// TIA Portal V16 export
// export: Created 2024-05-16T13:10:21.6108295Z, ExportSetting WithDefaults, DisplayName Totally Integrated Automation Portal, DisplayVersion V16, DisplayName TIA Portal Version Control Interface, DisplayVersion V16, DisplayName TIA Portal Openness, DisplayVersion V16, DisplayName STEP 7 Professional, DisplayVersion V16, DisplayName STEP 7 Safety, DisplayVersion V16, DisplayName WinCC Professional, DisplayVersion V16
DATA_BLOCK "DB22001_Dy_InstAnalogRead"   // DB22001
TITLE = Dynamic DB [INSTRUMENTATION] — Analog Instrument Read, Scale and Monitor
{ S7_Optimized_Access := 'TRUE' }
AUTHOR : M_Gledhill
FAMILY : Instrumentation
NAME : Dy_InstAnalogRead
VERSION : 3.0
// PRACTICAL SERIES AUTOMATION LIBRARY (PAL)   —   COPYRIGHT 2020 – M. GLEDHILL (MIT LICENCE)
//                   ———— ◆ ————
// FULL ONLINE DOCUMENTATION IS AVAILABLE AT: https://practicalseries.com/2001-pal/index.html
// stored: AutoNumber false, DBAccessibleFromOPCUA true, IsOnlyStoredInLoadMemory false, IsRetainMemResEnabled false, IsWriteProtectedInAS false, MemoryReserve 100
   VAR
      _DB_Header { ExternalAccessible := 'False'; ExternalVisible := 'False'; ExternalWritable := 'False'} : Array[0..79] of Bool;   // Dynamic DB [INSTRUMENTATION] — Analog Instrument Read, Scale and Monitor
      __________0000_0 { ExternalAccessible := 'False'; ExternalVisible := 'False'; ExternalWritable := 'False'} : Bool := false;
      __________0000_1 { ExternalAccessible := 'False'; ExternalVisible := 'False'; ExternalWritable := 'False'} : Bool := false;   // ▀▀▀▀ DB CURRENT REVISION
      revInfo { ExternalWritable := 'False'; S7_SetPoint := 'True'} : "UT01000_St_SysRevision";   // Revision information
      __________0010_0 { ExternalAccessible := 'False'; ExternalVisible := 'False'; ExternalWritable := 'False'} : Bool := false;
      __________0010_1 { ExternalAccessible := 'False'; ExternalVisible := 'False'; ExternalWritable := 'False'} : Bool := false;   // ▀▀▀▀ ANALOG INSTRUMENTS
      FIC101 { S7_SetPoint := 'True'} : "UT22001_Dy_InstAnalogRead";   // Filter 1 outlet flow
   END_VAR
BEGIN
   // _DB_Header[0] : ▄▄▄▄▄▄▄▄▄▄▄▄▄▄▄▄▄▄▄▄▄▄▄▄▄▄▄▄▄▄▄▄▄ ＳＴＡＮＤＡＲＤ ▄▄
   // _DB_Header[2] : TITLE: INSTRUMENTATION — ANALOG INSTRUMENT READ, SCALE AND MONITOR
   // _DB_Header[4] : ▀▀▀▀▀▀▀▀▀▀▀▀▀▀▀▀▀▀▀▀▀▀▀▀▀▀▀▀▀▀▀▀▀▀▀▀▀▀▀▀▀▀▀▀
   // _DB_Header[5] : TYPE: DYNAMIC
   // _DB_Header[6] : ▄▄▄▄▄▄▄▄▄▄▄▄▄▄▄▄▄▄▄▄▄▄▄▄▄▄▄▄▄▄▄▄▄▄▄▄▄▄▄▄▄▄▄▄
   // _DB_Header[8] : This is the dynamic data block associated with the standard analog instrument read
   // _DB_Header[9] : block:
   // _DB_Header[10] : FC02001_StdInstAnalog
   // _DB_Header[12] : The dynamic data holds the current scaled value of the instrument, along with
   // _DB_Header[13] : any alarms, warnings or faults.
   // _DB_Header[15] : Each instrument is given the user data type:
   // _DB_Header[16] : UT22001_Dy_InstAnalog
   // _DB_Header[17] : This holds the full set of static configuration data for the instrument.
   // _DB_Header[19] : ━━━ ⬙⬙⬙⬙⬙⬙ ━━━
   // _DB_Header[21] : ▄▄▄▄▄▄▄▄▄▄▄▄▄▄▄▄▄▄▄▄▄▄▄▄▄▄▄▄▄▄▄▄▄▄▄▄▄▄▄▄▄▄▄▄
   // _DB_Header[22] : MODIFICATION HISTORY
   // _DB_Header[24] : This is a summary of the recent software modifications made to this block (most recent at top)
   // _DB_Header[26] : ―――――――――――――――――――――――――――――――――――――――――――
   // _DB_Header[27] : DATE REVISION MASTER BRANCH DEV
   // _DB_Header[28] : (nnn.amm) COMMIT TAG (Base ---> Merge) BRANCH Author
   // _DB_Header[29] : ———————————————————————————————————————————
   // _DB_Header[30] : 2024.05.16 003.000 D0017A-000.105 D0017 D0018 None M. Gledhill
   // _DB_Header[31] : FC02001 — RELEASED FOR USE
   // _DB_Header[32] : Merge back to master branch
   // _DB_Header[34] : 2024.05.11 002.801 D0017A-000.104 D0017 N/A D017A M. Gledhill
   // _DB_Header[35] : RAW_ANALOG changed to AI_RAW_SIGNAL
   // _DB_Header[36] : AI_RAW_DATA and AI_SCALE_DATA added and
   // _DB_Header[37] : copied to DYNAMIC_DATA (see db00801 SMDS)
   // _DB_Header[39] : 2022.04.16 002.000 D0011 D0010 D0011 None M. Gledhill
   // _DB_Header[40] : FC02001 — RELEASED FOR USE
   // _DB_Header[41] : Merge back to master branch
   // _DB_Header[43] : 2022.04.11 001.801 D0010A-000.801 D0010 N/A D010A M. Gledhill
   // _DB_Header[44] : Released for test (SCV)
   // _DB_Header[46] : 2022.04.08 001.102 D0010A-000.104 D0010 N/A D010A M. Gledhill
   // _DB_Header[47] : Comments updated
   // _DB_Header[49] : 2022.04.05 001.101 D0010A-000.103 D0010 N/A D010A M. Gledhill
   // _DB_Header[50] : Over and under range based on scaled signal
   // _DB_Header[51] : INFO_TYPE, cal_OR_Abs and cal_UR_Abs added
   // _DB_Header[52] : Comments updated and standardised
   // _DB_Header[53] : UDT variable names standardised
   // _DB_Header[55] : 2021.05.26 001.000 D0008 D0006 D0008 None M. Gledhill
   // _DB_Header[56] : FC02001 — RELEASED FOR USE
   // _DB_Header[57] : Merge back to master branch
   // _DB_Header[59] : 2021.05.24 000.801 D0006B-000.801 D0006 N/A D0006B M. Gledhill
   // _DB_Header[60] : FC02001 — Released for SMT
   // _DB_Header[62] : 2021.05.18 000.101 D0006B-000.101 D0006 N/A D0006B M. Gledhill
   // _DB_Header[63] : FC02001 Migration to VCS
   // _DB_Header[64] : ———————————————————————————————————————————
   // _DB_Header[65] : Where: nnn = Major revision
   // _DB_Header[66] : a = Type (1-7 Development, 8 Proving, 9 Qualification, 0 Release)
   // _DB_Header[67] : mm = Minor revision (must be 00 if a = 0)
   // _DB_Header[68] : Block properties version number should be set to nn.a (only one decimal place)
   // _DB_Header[70] : ██████████████ █ █ █ █ END █ █ █ █ ██████████████
   revInfo.REV_BLOCK := 'DB22001';
   revInfo.REV_NUMBER := '003.000';
   revInfo.REV_DATE := '2024-05-16';
   revInfo.REV_AUTHOR := 'M. Gledhill';
   FIC101.revInfo.REV_BLOCK := 'DB22001';
   FIC101.revInfo.REV_NUMBER := '000.801';
   FIC101.revInfo.REV_DATE := '2021-05-24';
   FIC101.revInfo.REV_AUTHOR := 'M. Gledhill';
END_DATA_BLOCK
